// TIA Portal V21 export
DATA_BLOCK "Fronte"   // DB3
{ S7_Optimized_Access := 'TRUE' }
// stored: MemoryReserve 100
   VAR RETAIN
      F : Array[0.."K_NumFrontiSalitaDiscesa"] of Struct
         Dati : Struct
            MemStatoPrec : Bool;
         END_STRUCT;
         Out : Struct
            StatoFronte : Bool;
         END_STRUCT;
      END_STRUCT;
   END_VAR
BEGIN
   F[0].Dati.MemStatoPrec := FALSE;
   F[0].Out.StatoFronte := FALSE;
END_DATA_BLOCK
